Staubli VAL3: start.pgx

program start()
begin
  call startingSockets()
  taskCreate "stateRobot", 1, statesRobot()
  taskCreate "moveRobot", 1, moveRobot()
  //taskCreate "moveRobot", 1, moveRobotSuc()
  taskCreate "screen", 1, pantalla()
end
